// TIA Portal V20 export
// export: Created 2025-12-01T14:57:43.9318292Z, ExportSetting None, DisplayName Totally Integrated Automation Portal, DisplayVersion V20 Update 3, DisplayName TIA Portal Openness, DisplayVersion V20 Update 3, DisplayName TIA Portal Version Control Interface, DisplayVersion V20 Update 3, DisplayName STEP 7 Professional, DisplayVersion V20 Update 3, DisplayName STEP 7 Safety, DisplayVersion V20 Update 2, DisplayName WinCC Basic/Comfort/Advanced, DisplayVersion V20 Update 3, DisplayName WinCC Professional, DisplayVersion V20 Update 3, DisplayName WinCC Unified, DisplayVersion V20 Update 3
FUNCTION "FC519_Buc_Lec_Scanners" : Void   // FC519, STL
{ S7_Optimized_Access := 'FALSE' }
AUTHOR : SSCC
NAME : 23062013
VERSION : 3.2
// stored: AutoNumber false
   VAR_TEMP
      NDB_TMP : Word;   // Num. DB Temporal
      PunteroTMP : DWord;   // Puntero Temporal
      DBNodosPresentes : UInt;   // DB De Nodos Presentes de la Red
      RedActual : UInt;   // Red actual de Lectura
      SCR_Actual : UInt;
      CNT_LectCiclo : UInt;   // Contador de lecturas en la Red
   END_VAR
BEGIN

NETWORK
TITLE = Inicializaciones
// --------------------------------------------------------------------------------------
// --- Incializar para recorrer las Redes de Escanneres

      L     1;
      T     #RedActual;



NETWORK
TITLE = Bucle de scanners
// --------------------------------------------------------------------------------------
// --- Inicializar datos de la Red de Scanners

_INI: NOP   0;

// --------------------------------------------------------------------------------------
// --- Comprobar si está configurada

      L     "DB911_Conf_Sistema_Scanners".Bucles_lectura_Scanner[#RedActual].NodoInicial;  // Si el Nodo Incial es cero
      L     0;  // No existe Scanner en la Red
      ==I;
      JC    _FIN;

// --------------------------------------------------------------------------------------
// --------------------------------------------------------------------------------------
// --- Lecturas de los Escaneres de la Red  (Bucle)

// --------------------------------------------------------------------------------------
// --- Incializaciones del Bucle

      L     0;  // --- Inicio Contador lecturas tradadas por ciclo
      T     #CNT_LectCiclo;

// --------------------------------------------------------------------------------------
// --- Comprobaciones del Nodo Actual a Comprobar

      L     "DB911_Conf_Sistema_Scanners".Bucles_lectura_Scanner[#RedActual].SCR_Actual;  // --- Comparamos con el numero de Scanneres definidos
      L     "DB911_Conf_Sistema_Scanners".Bucles_lectura_Scanner[#RedActual].NodoInicial;  //     Si estamos dentro de la Red de Scanners
      >=I;
      JC    ISRC;

      L     "DB911_Conf_Sistema_Scanners".Bucles_lectura_Scanner[#RedActual].NodoInicial;
      T     "DB911_Conf_Sistema_Scanners".Bucles_lectura_Scanner[#RedActual].SCR_Actual;  // --- Inicimos el Número de Scanner a tratar de 0..n

ISRC: L     "DB911_Conf_Sistema_Scanners".Bucles_lectura_Scanner[#RedActual].SCR_Actual;
      L     "DB911_Conf_Sistema_Scanners".Bucles_lectura_Scanner[#RedActual].NodoFinal;  // --- Comparamos con el numero de Scanners definidos
      <=I;  //     Si estamos en el ultimo ponemos al Inicio de la Red.
      JC    TIPO;  //    SPB   BSRC

      L     "DB911_Conf_Sistema_Scanners".Bucles_lectura_Scanner[#RedActual].NodoInicial;
      T     "DB911_Conf_Sistema_Scanners".Bucles_lectura_Scanner[#RedActual].SCR_Actual;  // --- Inicimos el Número de Scanner a tratar de 0..n


TIPO: SET;  // Comprobamos si es nodo profibus o profinet para hacer el diagnóstico dentro de la red
// -- si estamos en modo simulacion no hacemos ningún diagnostico de nodo
      SET;
      A     "Activar_Simulador";
      JC    comprobar_si_hay_etiqueta;

// -- Comprobamos el tipo de modelo para hacer el diagnostico del nodo
      L     "DB911_Conf_Sistema_Scanners".Bucles_lectura_Scanner[#RedActual].Modelo;
      L     DINT#5;
      >=I;
      JC    bucle_profinet;  // bucle de profinet



NETWORK
TITLE = Comprobacion de Nodos
//*******************************************************************************
// --- Comprobacion si el Nodo existe   (ZONA PROFIBUS)
// ZONA DE PROFIBUS QUEDA COMENTADA POR ESTAR CASI OBSOLETA
// DE QUERER ACTIVARLA OTRA VEZ, DESCOMENTAR LA ZONA MARCADA ENTRE INICIO Y FIN
//-- INICIO ZONA PROFIBUS 20200508

      L     #DBNodosPresentes;  // --- Formatea DB Errores Para poder Abrirlo
      T     #NDB_TMP;

      L     P#52.0;  // --- Direccion del Bit dentro del DB de Errores
      L     "DB911_Conf_Sistema_Scanners".Bucles_lectura_Scanner[#RedActual].SCR_Actual;  //     Bit del Nodo Presente (Actual)
      +D;
      L     1;
      -D;
      T     #PunteroTMP;

      OPN   DB [#NDB_TMP];  // --- Existe Nodo ?
      SET;
      A     DBX [#PunteroTMP];
      JC    Siguiente_Scanner;

      L     #PunteroTMP;  // --- Direccion del Bit dentro del DB de Errores
      L     128;  //     Bit del Error del Nodo (Actual)
      +D;
      T     #PunteroTMP;

      OPN   DB [#NDB_TMP];  // --- Nodo en Error ?
      SET;
      A     DBX [#PunteroTMP];
      JC    Siguiente_Scanner;

      JU    comprobar_si_hay_etiqueta;  // salta a la comprobación

//-- FIN ZONA PROFIBUS 20200508
//*******************************************************************************


//================================================================================
// --- Comprobacion si el Nodo existe   (ZONA PROFINET)
bucle_profinet:SET;

      L     "DB911_Conf_Sistema_Scanners".Bucles_lectura_Scanner[#RedActual].SCR_Actual;
      T     #SCR_Actual;

      SET;
      AN    "DB927_PNIODiag_Data".RED[1].NODO[#SCR_Actual].OK;
      JC    Siguiente_Scanner;

//================================================================================


NETWORK
TITLE = Comprobación de si existe etiqueta
// ------------------------------------------------------------------------------
// --- Mirar y Extraer la Eiqueta del Nodo Actual del Scanner
// --- Llamada a la lectura dependiendo de Modelo

comprobar_si_hay_etiqueta:NOP   0;



      L     "DB911_Conf_Sistema_Scanners".Bucles_lectura_Scanner[#RedActual].Modelo;  // --- Reparto por Modelo de Scanner
      JL    LSTX;

      JU    DATL;  // --- Modelo DataLogic profibus  (0)
      JU    SICK;  // --- Modelo SICK profibus      (1)
      JU    SICA;  // --- Modelo SICK para router alfanumérico  profibus  (2)
      JU    Siguiente_Scanner;  // --- RESERVA PROFIBUS
      JU    Siguiente_Scanner;  // --- RESERVA PROFIBUS
      JU    SICN;  // --- Modelo SICK para profinet (5) Añadido Nieves 17/08/16
      JU    SIAN;  // --- Modelo SICK ALFANUMERICO para profinet (6) Añadido Nieves 17/08/16
      JU    SILINT;  // MODELO SICK PARA ETIQUETAS ULINT (7)

LSTX: JU    Siguiente_Scanner;  // --- No definido


// ------------------------------------------------------------------------------
// --- Tratamiento de Scanner de Modelo DataLogic profibus

DATL: NOP   0;
//      CALL  "FC524_Form_Lec_Modelo_DL"
//         Red_Actual    :=#RedActual
//         Datos_Red     :=#Datos_Red
//         CNT_LectCiclo :=#CNT_LectCiclo

// en caso de que sea necesario recuperar la función,
// recoger de librería obsoletos scanners
      JU    Siguiente_Scanner;

// ------------------------------------------------------------------------------
// --- Tratamiento de Scanner de Modelo SICK profibus

SICK: NOP   0;
//  CALL  "FC525_Form_Lect_Modelo_SICK"
//         Red_Actual    :=#RedActual
//         Datos_Red     :=#Datos_Red
//         CNT_LectCiclo :=#CNT_LectCiclo

// en caso de que sea necesario recuperar la función,
// recoger de librería obsoletos scanners

      JU    Siguiente_Scanner;


// ------------------------------------------------------------------------------
// --- Tratamiento de Scanner de Modelo SICK para router alfanumérico profibus

SICA: NOP   0;

//   CALL  "FC526_Form_Lec_Modelo_SICK_ALF"
//         Red_Actual    :=#RedActual
//         Datos_Red     :=#Datos_Red
//         CNT_LectCiclo :=#CNT_LectCiclo

// en caso de que sea necesario recuperar la función,
// recoger de librería obsoletos scanners

      JU    Siguiente_Scanner;

// ------------------------------------------------------------------------------
// --- Tratamiento de Scanner de Modelo SICK profinet

SICN: SET;
      CALL  "FC527_Form_Lec_Modelo_SICK_PN"
      ( Numero_Red    := #RedActual,
        Datos_red     := "DB911_Conf_Sistema_Scanners".Bucles_lectura_Scanner[#RedActual],
        CNT_LectCiclo := #CNT_LectCiclo
      );

      JU    Siguiente_Scanner;


// ------------------------------------------------------------------------------
// --- Tratamiento de Scanner de Modelo SICK para router alfanumérico profinet


SIAN: SET;
      CALL  "FC528_Form_Lec_Mod_SICK_PN_ALF"
      ( Numero_Red    := #RedActual,
        Datos_Red     := "DB911_Conf_Sistema_Scanners".Bucles_lectura_Scanner[#RedActual],
        CNT_LectCiclo := #CNT_LectCiclo
      );


SILINT:SET;
      CALL  "FC529_Form_Lec_Modelo_SICK_PN_ULINT"
      ( Numero_Red    := #RedActual,
        Datos_red     := "DB911_Conf_Sistema_Scanners".Bucles_lectura_Scanner[#RedActual],
        CNT_LectCiclo := #CNT_LectCiclo
      );

      JU    Siguiente_Scanner;

// ------------------------------------------------------------------------------



NETWORK
TITLE = pasar al siguiente scanner

// ------------------------------------------------------------------------------
// --- Maximas Lecturas de Ciclo en la Red

Siguiente_Scanner:NOP   0;
      L     #CNT_LectCiclo;  // --- Valida la cantidad Maxima de lecturas tratadas por ciclo
      L     "ROUT_Max_Lec_Ciclo";  // L     "DB911_Conf_Sistema_Router".Num_Max_Lec_Ciclo
      >=I;
      JC    FSRC;

// ------------------------------------------------------------------------------------------------
// --- Nodo Siguiente de la Red

      L     1;
      L     "DB911_Conf_Sistema_Scanners".Bucles_lectura_Scanner[#RedActual].SCR_Actual;  // Incrementamos el scanner que debe de ser tratado
      +I;
      T     "DB911_Conf_Sistema_Scanners".Bucles_lectura_Scanner[#RedActual].SCR_Actual;

      SET;
      L     "DB911_Conf_Sistema_Scanners".Bucles_lectura_Scanner[#RedActual].SCR_Actual;  // Si estamos en el ultimo salimos del Bucle
      L     "DB911_Conf_Sistema_Scanners".Bucles_lectura_Scanner[#RedActual].NodoFinal;  // Comparamos con el numero de Scanners definidos
      <=I;
      JC    TIPO;  //  SPB   BSRC

// ------------------------------------------------------------------------------------------------
// --- Final del Bucle

FSRC: NOP   0;


// --------------------------------------------------------------------------------------
// --------------------------------------------------------------------------------------
// --------------------------------------------------------------------------------------
// --------------------------------------------------------------------------------------
// --------------------------------------------------------------------------------------
// --------------------------------------------------------------------------------------



// --------------------------------------------------------------------------------------
// --- Siguiente Red

      L     #RedActual;  // Ultima Red a Testear
      L     5;  // Red --> 1...5
      ==I;
      JC    _FIN;

      L     #RedActual;  // Siguiente Red Scanneres
      L     1;
      +I;
      T     #RedActual;

      JU    _INI;  // A Testear Siguiente Red




NETWORK
TITLE = 
// --------------------------------------------------------------------------------------
// --- Final de la Funcion

_FIN: NOP   0;



END_FUNCTION
